# EPICS autosave request: caenN1470/caenN1470_settings.req
$(P)$(Q):UPDATE.SCAN
$(P)$(Q):UPDATECHAN.SCAN
